(* CODESYS project cyber-gprs.lib.source.20190613.project

Project tree, tasks and I/O mapping:
  MIC7001 : Changsha Xiangji-ARM Cortex A9(xilinx zynq7000)-linux, Changsha Xiangji Hiden Technology Co.Ltd, version 3.5.10.40
    application Application
      libraries: CAA Types Extern, 3.5.10.0 (CAA Technical Workgroup); VisuDialogs, * (System); CAA Real Time Clock Extern, 3.5.10.0 (CAA Technical Workgroup); CAA Callback Extern, 3.5.11.0 (CAA Technical Workgroup); CAA Can Low Level Extern, 3.5.11.0 (CAA Technical Workgroup); CAA Can Low Level Imp Extern, 3.5.11.0 (CAA Technical Workgroup); SysMem, 3.5.12.0 (System); CAA Net Base Services, 3.5.12.0 (CAA Technical Workgroup); CAA SerialCom, 3.5.12.0 (CAA Technical Workgroup); CAA File, 3.5.12.0 (CAA Technical Workgroup); CAA DTUtil Extern, 3.5.12.0 (CAA Technical Workgroup); SysFile, 3.5.9.0 (System); SysTypes2 Interfaces, * (System); Standard, * (System); cyber gpio, 3.5.10.40 (cyber); Util, * (System)
      task Task_gprs (cyclic, interval 20 ms, priority 10) calls prg_heartbeat
      global variables GVL
      GPRS/
        function block File_Read [ST]
        function Iccid_Get [ST]
        program prg_heartbeat [ST]
        function block fb_get_iccid [ST]
        function block fb_m26 [ST]
        function block fb_get_lac [ST]
        function fn_cyber_layer1 [ST]
        function fn_cyber_layer2 [ST]
        function fn_cyber_heartBeat [ST]
        function fn_sn_str_to_byte [ST]
      gprs_lib/
        function block Com_Read [ST]
        function block reset_gprs [ST]
        function block Udp_Config [ST]
        function block Udp_Init [ST]
        function block UDP_Read [ST]
        function block Udp_Write [ST]
    IoDrvMIC7001 : IoDrvMIC7001, Cyber-MI, version 18.11.1
        unmapped channels: Ai00@C16, Ai01@C28, Ai02@C17, Ai03@C29, Ai04@C30, Ai05@C19, Ai06@C31, Ai07@C20, Ai08@C18, Ai09@D18, Ai10@D20, Ai11@D31, Ai12@D19, Ai13@D30, Ai14@D29, Ai15@D17, Ai16@D28, Ai17@D16, Ai18-Do00@C25, Ai19-Do01@C24, Ai20-Do02@C13, Ai21-Do03@C01, Ai22-Do04@C03, Ai23-Do05@C04, Ai24-Do06@C05, Ai25-Do07@C06, Ai26-Do08@C08, Ai27-Do09@C09, Ai28-Do10@C10, Ai29-Do11@C11, Ai30-Do12@D34, Ai31-Do13@D35, Ai32-Do14@D23, Ai33-Do15@D12, Ai34-Do16@D10, Ai35-Do17@D09, Ai36-Do18@D08, Ai37-Do19@D07, Ai38-Do20@D05, Ai39-Do21@D04,
          Ai40-Do22@D03, Ai41-Do23@D02, Ai42-Do24@C23, Ai43-Do25@C35, Ai44-Do26@D24, Ai45-Do27@D13, Ai46-Ao00@C22, Ai47-Ao01@D14, Ai48_Pi02, Ai49_Out5V, Ai50_VCC, Ai51_VCC_L, Ai52_VCC_R, Ai53_Pwm-i0, Ai54_Pwm-i1, Ai55_Pwm-i2, Ai56_Pwm-i3, Ai57_CPU-T, Ai58_G-x, Ai59_G-y, Ai60_G-z, Ai61-reserved, Ai62-IO-cntr, Ai63-CDS-cntr, Di00-Ai00@C16, Di01-Ai01@C28, Di02-Ai02@C17, Di03-Ai03@C29, Di04-Ai04@C30, Di05-Ai05@C19, Di06-Ai06@C31, Di07-Ai07@C20, Di08-Ai08@C18, Di09-Ai09@D18, Di10-Ai10@D20, Di11-Ai11@D31, Di12-Ai12@D19, Di13-Ai13@D30, Di14-Ai14@D29, Di15-Ai15@D17,
          Di16-Ai16@D28, Di17-Ai17@D16, Di18-Ai18@C25, Di19-Ai19@C24, Di20-Ai20@C13, Di21-Ai21@C01, Di22-Ai22@C03, Di23-Ai23@C04, Di24-Ai24@C05, Di25-Ai25@C06, Di26-Ai26@C08, Di27-Ai27@C09, Di28-Ai28@C10, Di29-Ai29@C11, Di30-Ai30@D34, Di31-Ai31@D35, Di32-Ai32@D23, Di33-Ai33@D12, Di34-Ai34@D10, Di35-Ai35@D09, Di36-Ai36@D08, Di37-Ai37@D07, Di38-Ai38@D05, Di39-Ai39@D04, Di40-Ai40@D03, Di41-Ai41@D02, Di42-Ai42@C23, Di43-Ai43@C35, Di44-Ai44@D24, Di45-Ai45@D13, Di46-Ai46@C22, Di47-Ai47@D14, Di48-Pi00@C15, Di49-Pi01@C14, Di50-Pi02@D22, Di51-Pi03@D21, Di52-reserved, Di53-reserved, Di54-reserved, Di55-reserved,
          Di56-reserved, Di57-reserved, Di58-reserved, Di59-reserved, Di60-reserved, Di61-reserved, Di62-reserved, Di63-reserved, Pi00-Di48@C15, Pi01-Di49@C14, Pi02-Di50@D22, Pi03-Di51@D21, Do00-Ai18@C25, Do01-Ai19@C24, Do02-Ai20@C13, Do03-Ai21@C01, Do04-Ai22@C03, Do05-Ai23@C04, Do06-Ai24@C05, Do07-Ai25@C06, Do08-Ai26@C08, Do09-Ai27@C09, Do10-Ai28@C10, Do11-Ai29@C11, Do12-Ai30@D34, Do13-Ai31@D35, Do14-Ai32@D23, Do15-Ai33@D12, Do16-Ai34@D10, Do17-Ai35@D09, Do18-Ai36@D08, Do19-Ai37@D07, Do20-Ai38@D05, Do21-Ai39@D04, Do22-Ai40@D03, Do23-Ai41@D02, Do24-Ai42@C23, Do25-Ai43@C35, Do26-Ai44@D24, Do27-Ai45@D13,
          Do28-Pwmi00@C33, Do29-Pwmi01@C34, Do30-Pwmi02@D25, Do31-Pwmi03@D26, PWM00@C25, PWM01@C24, PWM02@C13, PWM03@C01, PWM04@C03, PWM05@C04, PWM06@C05, PWM07@C06, PWM08@C08, PWM09@C09, PWM10@C10, PWM11@C11, PWM12@D34, PWM13@D35, PWM14@D23, PWM15@D12, PWM16@D10, PWM17@D09, PWM18@D08, PWM19@D07, PWM20@D05, PWM21@D04, PWM22@D03, PWM23@D02, PWM24@C23, PWM25@C35, PWM26@D24, PWM27@D13, PWM28-Pwmi00@C33, PWM29-Pwmi01@C34, PWM30-Pwmi02@D25, PWM31-Pwmi03@D26, PWM_I_0@C33, PWM_I_1@C34, PWM_I_2@D25, PWM_I_3@D26,
          Ao00-Ai46@C22, Ao01-Ai47@D14, LED_run, LED_err, LED_usr, ctrl_ai_raw, ctrl_adjust, ctrl_adj0, ctrl_adj1, ctrl_adj2, ctrl_adj3, ctrl_adj4
    SoftMotion General Axis Pool
  5ce3da45-db07-42e7-a21c-a00fff4ed8f6|C:\Users\Administrator\Desktop\robotview1.bmp
  5ce3da45-db07-42e7-a21c-a00fff4ed8f6|C:\Users\Administrator\Desktop\robotview2.bmp
  text list GlobalTextList
  5ce3da45-db07-42e7-a21c-a00fff4ed8f6|C:\Users\Administrator\Desktop\1129.bmp
  5ce3da45-db07-42e7-a21c-a00fff4ed8f6|C:\Users\Administrator\Desktop\robotview0.bmp
*)

// MIC7001/Application/GVL
VAR_GLOBAL
	
END_VAR

// MIC7001/Application/GPRS/prg_heartbeat
PROGRAM prg_heartbeat
VAR_OUTPUT
	lock_state :INT := 0;
	unlock_state :INT := 0;
	lock_unlock_level :INT := 0;
	delay_time :INT := 0;
END_VAR

VAR
	is_inited :BOOL := FALSE;
	g_m26:fb_m26;
	udp_handle :CAA.HANDLE; 
	udp_write_fb:Udp_Write;
	udp_read_fb:Udp_Read;
	file_read_fb:File_Read;
	com_read_fb :Com_Read;


	size :CAA.SIZE;	
	Writebuffer: 			ARRAY[1..200] OF BYTE;
	Readbuffer: 			ARRAY[0..1499] OF BYTE;
	ReadbufferStr: STRING;
	atcState :INT := 0;
	
	writeUdpState :INT := 0;
	readUdpState :INT := 0;
	
	i :INT;
	count :INT := 0;
	
	rtc_fb: RTC;
	dtu_set_dt_fb: dtu.SetDateAndTime;
	
	sn_file_name :STRING := '/userapp/sn.txt';
	time_file_name :STRING := '/userapp/r_mins.txt';
	is_read :BOOL := FALSE;
	read_count :INT := 0;
	readFileState :INT := 0;
	ton_fb :TON;
	iccid_read_buffer :STRING;
	position :INT := -1;
	new_date:DT;
	get_iccid:fb_get_iccid;
	get_lac:fb_get_lac;
	iStat :UINT := 0;
	lac : STRING(4) := '0000';
	ci : STRING(4) := '0000';
	lenHearBeat:UINT;
	dataHearBeat:ARRAY[0..255] OF BYTE;
	ton_hb:ton; //heartbeat timer 
	bReturn:BOOL;
	lenLayer2:UINT;
	dataLayer2:ARRAY[0..255] OF BYTE;
	lenLayer1:UINT;
	lenRecvLayer1:UINT := 1500;
	dataLayer1:ARRAY[0..255] OF BYTE;
	bSN :ARRAY[0..6] OF BYTE;
	sub_str:STRING(8);
	num :UINT;
	lenHeartBeat: UINT;
	sn: STRING;
	work_time: UDINT;
	dataIndex :UINT := 0;
	cntr_lac:UINT := 0;
	cntr_iccid:UINT := 0;
	
	recv_size :CAA.SIZE;
END_VAR

CASE iStat OF
0:
	g_m26(enable := TRUE, ipaddr := '47.107.240.29', port := 20861);  //共用的基础模块，只要有一个地方调用即可	
	IF g_m26.xDone THEN
		iStat := 1;
	END_IF


1:  // read iccid
	get_iccid(xExecute := FALSE);
	iStat := 2;
	cntr_iccid := 0;
	
2:
	get_iccid(xExecute := TRUE, m26_handle := g_m26.handle_m26);
	IF get_iccid.xDone THEN
		iccid_read_buffer := get_iccid.iccid;
		iStat := 10;
	END_IF
	cntr_iccid := cntr_iccid + 1;
	IF cntr_iccid > 600 THEN   // 1 min
		iStat := 1;
	END_IF
	
10: //read sn
	file_read_fb(file_name := sn_file_name);
	IF file_read_fb.isRead THEN
		sn := file_read_fb.sReadLine;
		iStat := 15;
	END_IF
	
15:
	get_lac(xExecute := FALSE);	
	iStat := 20;
	cntr_lac := 0;
	
20:
	get_lac(xExecute := TRUE, m26_handle := g_m26.handle_m26);
	IF get_lac.xDone THEN
		lac := get_lac.lac;
		ci := get_lac.ci;
		iStat := 30;
	END_IF
	cntr_lac := cntr_lac + 1;
	IF cntr_lac > 200 THEN
		iStat := 0;
	END_IF
	
30:
	file_read_fb(file_name := time_file_name);
	IF file_read_fb.isRead THEN
		work_time := STRING_TO_UDINT(file_read_fb.sReadLine);
		iStat := 100;
	END_IF
	
100:
	ton_fb(IN := TRUE, PT := T#60S);
	IF (ton_fb.Q) THEN
		ton_fb(IN := FALSE, PT := T#60S);
		iStat := 200;
	END_IF
	
200:
	bReturn := fn_cyber_heartBeat(	  //填充第三层：心跳帧
						lac_str := lac, 
						cid_str := ci, 
						ccid_str := iccid_read_buffer, 
						mins := work_time, 
						clientCode := 1, 
						machineCode := 1, 
						pLenOut := ADR(lenHearBeat), 
						pDataOut := ADR(dataHearBeat));
	IF NOT bReturn THEN
		RETURN;
	ELSE
		iStat := 300;
	END_IF;

300:
	dataIndex := dataIndex + 1;
	bReturn := fn_cyber_layer2( //填充第二层，数据层
						dataType := 1,
						paraId := 0,
						dataIndex := dataIndex,
						ver := 1,
						res1 := 0,
						LenIn := lenHearBeat,
						pDataIn := ADR(dataHearBeat),
						pLenOut := ADR(lenLayer2),
						pDataOut := ADR(dataLayer2));
						
	IF NOT bReturn THEN
		RETURN;
	ELSE
		iStat := 400;
	END_IF;
	
400:
	bSN := fn_sn_str_to_byte(sn);
	bReturn := fn_cyber_layer1(    //填充第一层，设备层
						sn := ADR(bSN),
						ver := 1,
						lenIn := lenLayer2,
						pDataIn := ADR(dataLayer2),
						pLenOut := ADR(lenLayer1),
						pDataOut := ADR(dataLayer1));
	IF NOT bReturn THEN
		RETURN;
	ELSE
		udp_write_fb(xExecute := FALSE);
		iStat := 500;
	END_IF;
		
	
500:
	udp_write_fb(xExecute := TRUE, com := g_m26.handle_m26, buffer := ADR(dataLayer1), size := lenLayer1);
	IF udp_write_fb.xDone THEN
		udp_write_fb(xExecute := FALSE);
		udp_read_fb(xExecute := FALSE);
		iStat := 600; 
	END_IF
	
	IF udp_write_fb.xError THEN  
		udp_write_fb(xExecute := FALSE);
		iStat := 15; 
	END_IF
	
	
600:
	udp_read_fb(xExecute := TRUE, com := g_m26.handle_m26, buffer := ADR(Readbuffer), rsize := sizeof(Readbuffer));
	IF udp_read_fb.xDone THEN  //接收到数据
	 	recv_size := udp_read_fb.size;
		udp_read_fb(xExecute := FALSE);
		iStat := 15; //read mins and lca again
		IF recv_size = 26 THEN
			lock_state := BYTE_TO_INT(Readbuffer[20]);
			unlock_state := BYTE_TO_INT(Readbuffer[21]);
			lock_unlock_level := BYTE_TO_INT(Readbuffer[22]);
			delay_time := BYTE_TO_INT(Readbuffer[23]);
		END_IF
	END_IF
	
	IF udp_read_fb.xError THEN  //接收到数据
		udp_read_fb(xExecute := FALSE);
		recv_size := 0;
		iStat := 15; //read mins and lca again
	END_IF

END_CASE

RETURN;

END_PROGRAM

// MIC7001/Application/GPRS/fn_cyber_heartBeat
FUNCTION fn_cyber_heartBeat : bool
VAR_INPUT
	lac_str:STRING(4);
	cid_str:STRING(4);
	ccid_str:STRING(21);
	mins:UDINT;
	clientCode:UINT;
	machineCode:UINT;
	pLenOut:POINTER TO UINT;
	pDataOut:POINTER TO BYTE;
END_VAR
VAR
	index: UINT;
	data_uint: UINT;
	data_byte_array:ARRAY[0..9] OF BYTE;
	i: INT;
END_VAR

fn_cyber_heartBeat := FALSE;

index := 0;
data_uint := STRING_TO_UINT(concat('16#',lac_str));
pDataOut[index] := ANY_TO_BYTE(data_uint/256);
index := index + 1;

pDataOut[index] := ANY_TO_BYTE(data_uint MOD 256);
index := index + 1;

data_uint := STRING_TO_UINT(concat('16#',cid_str));
pDataOut[index] := ANY_TO_BYTE(data_uint/256);
index := index + 1;

pDataOut[index] := ANY_TO_BYTE(data_uint MOD 256);
index := index + 1;

data_byte_array := Iccid_Get(ccid_str);
FOR i := 0 TO 9 DO
	pDataOut[index] := data_byte_array[i];
	index := index + 1;
END_FOR

pDataOut[index] := ANY_TO_BYTE(mins/256/256/256);
index := index + 1;

pDataOut[index] := ANY_TO_BYTE(mins/256/256);
index := index + 1;

pDataOut[index] := ANY_TO_BYTE(mins/256);
index := index + 1;

pDataOut[index] := ANY_TO_BYTE(mins);
index := index + 1;

pDataOut[index] := ANY_TO_BYTE(clientCode/256);
index := index + 1;

pDataOut[index] := ANY_TO_BYTE(clientCode);
index := index + 1;

pDataOut[index] := ANY_TO_BYTE(machineCode/256);
index := index + 1;

pDataOut[index] := ANY_TO_BYTE(machineCode);
index := index + 1;

pLenOut^ := index;

fn_cyber_heartBeat := TRUE;

END_FUNCTION

// MIC7001/Application/GPRS/Iccid_Get
FUNCTION Iccid_Get : ARRAY[0..9] OF BYTE
VAR_INPUT
	iccd :STRING;
END_VAR
VAR
	iccid_code :ARRAY[0..9] OF BYTE;
	
	byteHigh :BYTE := 0;
	byteLow :BYTE := 0;
	dstLen :INT := 0;
	
	srcIndex :INT := 0;
	bytesIndex :INT := 0;
	sub_str:STRING(32);
END_VAR

dstLen := len(iccd) / 2;

sub_str := iccd;
FOR bytesIndex := 0 TO dstLen - 1 DO
	iccid_code[bytesIndex] := BYTE_TO_BCD(STRING_TO_BYTE(left(sub_str,2)));	
	sub_str := delete(sub_str,2,1);
END_FOR

Iccid_Get := iccid_code;

END_FUNCTION

// MIC7001/Application/GPRS/fn_cyber_layer2
FUNCTION fn_cyber_layer2 : bool
VAR_INPUT
	dataType : BYTE := 0;
	paraId :BYTE := 0;
	dataIndex : UINT := 0;
	ver :BYTE := 1;
	res1 :BYTE := 0;
	LenIn :UINT := 0;
	pDataIn :POINTER TO BYTE;
	pLenOut :POINTER TO UINT;
	pDataOut :POINTER TO BYTE;
END_VAR
VAR
	i:UINT:= 0;
	index:UINT := 0;
END_VAR

fn_cyber_layer2 := FALSE;

index := 0;
pDataOut[index] := dataType;
index := index + 1;

pDataOut[index] := paraId;
index := index + 1;

pDataOut[index] := ANY_TO_BYTE(dataIndex/256);
index := index + 1;

pDataOut[index] := ANY_TO_BYTE(dataIndex MOD 256);
index := index + 1;

pDataOut[index] := ver;
index := index + 1;

pDataOut[index] := res1;
index := index + 1;

pDataOut[index] := ANY_TO_BYTE(LenIn/256);
index := index + 1;

pDataOut[index] := ANY_TO_BYTE(LenIn MOD 256);
index := index + 1;

FOR i := 0 TO LenIn-1 DO
	pDataOut[index] := pDataIn[i];
	index := index + 1;
END_FOR

pLenOut^ := index;

fn_cyber_layer2 := TRUE;
RETURN;

END_FUNCTION

// MIC7001/Application/GPRS/fn_sn_str_to_byte
FUNCTION fn_sn_str_to_byte : ARRAY[0..6] OF BYTE
VAR_INPUT
	sn:STRING(16);
END_VAR
VAR
	i: INT;
	bSN: ARRAY[0..6] OF BYTE;
	sub_str: STRING(255);
	num: UINT;
	bcd: UINT;
END_VAR

// 1.2 12
sub_str := mid(sn, 2, 4);
bcd := STRING_TO_UINT(sub_str);
bcd := (bcd / 10) *16 + (bcd MOD 10);
bSN[0] := UINT_TO_BYTE(bcd);

// 1.3 34
sub_str := mid(sn, 2, 6);
bcd := STRING_TO_UINT(sub_str);
bcd := (bcd / 10) *16 + (bcd MOD 10);
bSN[1] := UINT_TO_BYTE(bcd);

// 1.4 56
sub_str := mid(sn, 2, 8);
bcd := STRING_TO_UINT(sub_str);
bcd := (bcd / 10) *16 + (bcd MOD 10);
bSN[2] := UINT_TO_BYTE(bcd);

// 1.5 78
sub_str := mid(sn, 2, 10);
bcd := STRING_TO_UINT(sub_str);
bcd := (bcd / 10) *16 + (bcd MOD 10);
bSN[3] := UINT_TO_BYTE(bcd);

// 1.6 1234
sub_str := mid(sn, 2, 12);
bcd := STRING_TO_UINT(sub_str);
bcd := (bcd / 10) *16 + (bcd MOD 10);
bSN[4] := UINT_TO_BYTE(bcd);

sub_str := mid(sn, 2, 14);
bcd := STRING_TO_UINT(sub_str);
bcd := (bcd / 10) *16 + (bcd MOD 10);
bSN[5] := UINT_TO_BYTE(bcd);

fn_sn_str_to_byte := bSN;

END_FUNCTION

// MIC7001/Application/GPRS/fn_cyber_layer1
FUNCTION fn_cyber_layer1 : bool
VAR_INPUT
	sn:POINTER TO BYTE;
	ver:BYTE := 0;
	lenIn:UINT := 0;
	pDataIn:POINTER TO BYTE;
	pLenOut:POINTER TO UINT ;
	pDataOut: POINTER TO BYTE;
END_VAR
VAR
	i:UINT;
	index:UINT;
	checksum:UINT;
	res1 :BYTE := 0;
	res2 :BYTE := 0;
	res3 :BYTE := 0;
END_VAR

fn_cyber_layer1 := FALSE;

index := 0;
checksum := 0;
FOR i := 0 TO 5 DO
	pDataOut[index] := sn[i];
	index := index+1;
	checksum := checksum + sn[i];
END_FOR

pDataOut[index] := ver;
index := index+1;
checksum := checksum + ver;

pDataOut[index] := res1;
index := index+1;
checksum := checksum + res1;

pDataOut[index] := res2;
index := index+1;
checksum := checksum + res2;

pDataOut[index] := res3;
index := index+1;
checksum := checksum + res3;

pDataOut[index] := ANY_TO_BYTE(lenIn/256);
index := index+1;
checksum := checksum + ANY_TO_BYTE(lenIn/256);

pDataOut[index] := ANY_TO_BYTE(lenIn MOD 256);
index := index+1;
checksum := checksum + ANY_TO_BYTE(lenIn MOD 256);

FOR i := 0 TO lenIn-1 DO
	pDataOut[index] := pDataIn[i];
	index := index+1;	
	checksum := checksum + pDataIn[i];
END_FOR

pDataOut[index] := ANY_TO_BYTE(checksum/256);
index := index+1;

pDataOut[index] := ANY_TO_BYTE(checksum MOD 256);
index := index+1;

pLenOut^ := index;

fn_cyber_layer1 := TRUE;

END_FUNCTION

// MIC7001/Application/GPRS/fb_m26
FUNCTION_BLOCK fb_m26
VAR_INPUT
	enable :BOOL := FALSE;
	ipaddr :STRING(32);
	port :UINT;
END_VAR
VAR_OUTPUT
	xBusy :BOOL := FALSE;
	xError :BOOL := FALSE;
	xDone :BOOL := FALSE;
	handle_m26 :CAA.HANDLE; 
END_VAR
VAR
	udp_init:Udp_Init;
	iStat :UINT := 0;
END_VAR

IF NOT enable THEN
	xBusy := FALSE;
	xError := FALSE;
	handle_m26 := 0;
	RETURN;
END_IF

CASE iStat OF
0:
	udp_init(xExecute := FALSE, ip_addr := ipaddr, port := port);
	udp_init.xExecute := TRUE;
	iStat := 10;
	
10:
	IF udp_init.xDone THEN
		xBusy := TRUE;
		handle_m26 := udp_init.udp_handle;
		iStat := 100;
	ELSIF udp_init.xError THEN
		iStat := 200;
	END_IF	

100:
	xDone:= TRUE;
	
200:
	xError := TRUE;

END_CASE


udp_init(ip_addr := ipaddr, port := port);

END_FUNCTION_BLOCK

// MIC7001/Application/gprs_lib/Udp_Init
FUNCTION_BLOCK Udp_Init
VAR_INPUT
	xExecute:BOOL := FALSE;
	ip_addr:STRING;
	port:UINT;
END_VAR
VAR_OUTPUT
	xDone :BOOL := FALSE;
	xError :BOOL := FALSE;
	xBusy :BOOL := FALSE;
	
	udp_handle :CAA.HANDLE; 
END_VAR
VAR
	udp_config_fb :Udp_Config;
	ComWrite: COM.Write;
	ComRead: COM.Read;	
	com_handle: CAA.HANDLE;
	init_start :DWORD := 0;
	iStat: INT := 0;
END_VAR

init_start := %ID48;
IF (init_start > 0) THEN
	RETURN;
END_IF

IF NOT xExecute THEN
	xDone := FALSE;
	xError := FALSE;
	xBusy := FALSE;
	iStat := 0;
	RETURN;
END_IF

CASE iStat OF
0:
	udp_config_fb(xExecute := FALSE,ip_addr := ip_addr, port := port, com_hand := com_handle); 
	iStat := 10;
	xBusy := TRUE;
10:
	udp_config_fb.xExecute := TRUE;
	IF udp_config_fb.xDone  THEN
		iStat := 100;
		xDone := TRUE;
		xBusy := FALSE;
		udp_handle := com_handle;
		ComWrite(xExecute := FALSE, hCom:= com_handle);
		ComRead(xExecute := FALSE, hCom:= com_handle);		
	ELSIF udp_config_fb.xError THEN
		xError := TRUE;
		iStat := 200;
	END_IF	
100: //succ

200: //error

END_CASE

udp_config_fb(ip_addr := ip_addr, port := port, com_hand := com_handle);

END_FUNCTION_BLOCK

// MIC7001/Application/gprs_lib/Udp_Config
FUNCTION_BLOCK Udp_Config
VAR_INPUT
	xExecute : BOOL := FALSE;
	ip_addr:STRING;
	port:UINT;
END_VAR
VAR_IN_OUT
	com_hand: CAA.HANDLE;
END_VAR
VAR_OUTPUT
	xDone : BOOL := FALSE;
	xError :BOOL := FALSE;
	xBusy : BOOL := FALSE;
END_VAR
VAR
	ton_fb :TON;
	Com1Params: 			ARRAY [1..7] OF COM.PARAMETER;	(* Settings to communicate with 
the COM Port *)
	ComOpen: 				COM.Open;
	ComClose: 				COM.Close;
	ComWrite: 				COM.Write;
	ComRead: 				COM.Read;	
	Rcv_Cnt: 				CAA.SIZE;
	xCom1CloseError: 		BOOL;
	xCom1WriteError: 		BOOL;
	xCom1ReadError: 		BOOL;
	uiComState: INT := 0;
	ComID:USINT:=6;

	position :INT := 0;
	at_cmd :STRING := 'AT$r';
	at_buffer :STRING;
	ate0_cmd :STRING := 'ATE0$r';
	ate0_buffer :STRING;
	cpin_cmd :STRING := 'AT+CPIN?$r';
	cpin_buffer :STRING;
	csq_cmd :STRING := 'AT+CSQ$r';
	csq_buffer :STRING;
	creg_cmd :STRING := 'AT+CREG?$r';
	creg_buffer :STRING;
	cgreg_cmd :STRING := 'AT+CGREG?$r';
	cgreg_buffer :STRING;
	qindi_cmd :STRING := 'AT+QINDI=1$r';
	qindi_buffer :STRING;     
	qimode_cmd :STRING := 'AT+QIMODE=0$r';
	qimode_buffer :STRING;     
	qifgcnt_cmd :STRING := 'AT+QIFGCNT=0$r';
	qifgcnt_buffer :STRING;
	qimux_cmd :STRING := 'AT+QIMUX=0$r';
	qimux_buffer :STRING;
	qicsgp_cmd :STRING := 'AT+QICSGP=1,$"CMNET$"$r';
	qicsgp_buffer :STRING;
	qideact_cmd :STRING := 'AT+QIDEACT$r';
	qideact_buffer :STRING;
	qiregapp_cmd :STRING := 'AT+QIREGAPP$r';
	qiregapp_buffer :STRING;
	qiact_cmd :STRING := 'AT+QIACT$r';
	qiact_buffer :STRING;
	qilocip_cmd :STRING := 'AT+QILOCIP$r';
	qilocip_buffer :STRING;
	qiopen_cmd :STRING := 'AT+QIOPEN=$"UDP$",$"';
	qiopen_buffer :STRING;
	
	qntp_cmd: STRING := 'AT+QNTP=$"s1a.time.edu.cn$"$r';
	qntp_buffer: STRING;
	qnitz_cmd: STRING := 'AT+QNITZ=1$r';	//启用同步网络时间
	qnitz_buffer :STRING;
	ctzu_cmd: STRING := 'AT+CTZU=1$r';
	ctzu_buffer: STRING;
	qlts_cmd: STRING := 'AT+QLTS$r';
	qlts_buffer: STRING;
	cclk_cmd: STRING := 'AT+CCLK?$r';
	cclk_buffer: STRING;
	
	NewDT : DT;
	NewDTS : STRING;
	NewDTSZH : STRING;
	dtu_set_dt_fb: dtu.SetDateAndTime;
	dtu_set_zone_fb: dtu.SetTimeZoneInformation;
	zone: RTCLK.TIME_ZONE_INFO;
	year: int;
	
	//dtu_get_zone_fb: dtu.GetTimeZoneInformation;
	//zone1: RTCLK.TIME_ZONE_INFO;

	loop_in_count :INT := 0;
	loop_out_count :INT := 0;
	loop_count :INT := 0;
	connect_cnt :INT := 0;
	reset_gprs_fb :reset_gprs;
END_VAR

IF NOT xExecute THEN
	xDone := FALSE;
	xError := FALSE;
	xBusy := FALSE;
	uiComState := 0;
	RETURN;
END_IF

CASE uiComState OF
	0:
	Com1Params[1].udiParameterId := COM.CAA_Parameter_Constants.udiPort;
	Com1Params[1].udiValue := ComID; 
	Com1Params[2].udiParameterId := COM.CAA_Parameter_Constants.udiBaudrate;
	Com1Params[2].udiValue := 115200;
	Com1Params[3].udiParameterId := COM.CAA_Parameter_Constants.udiParity;
	Com1Params[3].udiValue := INT_TO_UINT(COM.PARITY.NONE);
	Com1Params[4].udiParameterId := COM.CAA_Parameter_Constants.udiStopBits;
	Com1Params[4].udiValue := INT_TO_UINT(COM.STOPBIT.ONESTOPBIT);
	Com1Params[5].udiParameterId := COM.CAA_Parameter_Constants.udiTimeout;
	Com1Params[5].udiValue := 0;
	Com1Params[6].udiParameterId := COM.CAA_Parameter_Constants.udiByteSize;
	Com1Params[6].udiValue := 8;
	Com1Params[7].udiParameterId := COM.CAA_Parameter_Constants.udiBinary;
	Com1Params[7].udiValue := 0;					
	ComOpen(xExecute := TRUE, usiListLength:=UINT_TO_USINT(SIZEOF(Com1Params)/SIZEOF(COM.PARAMETER)),pParameterList:= ADR(Com1Params),hCom=> com_hand);			
	IF ComOpen.xError THEN
		uiComState := 32767;
	ELSIF ComOpen.xDone THEN
		uiComState := 1;
		com_hand := ComOpen.hCom;
		ComWrite(xExecute := FALSE,hCom:= com_hand);	
		ComRead(xExecute := FALSE,hCom:= com_hand);
	END_IF
	
	1:  // write "AT\r"
	ComWrite(xExecute := TRUE,hCom:= com_hand,pBuffer:= ADR(at_cmd),szSize:=len(at_cmd));		
	IF ComWrite.xError THEN
		uiComState := 32767;
	END_IF
	IF ComWrite.xDone THEN
		ComWrite(xExecute := FALSE, hCom:= com_hand);
		uiComState := 2;
	END_IF
	
	2:
	ton_fb(IN := TRUE, PT := TIME#300MS);
	IF (ton_fb.Q) THEN
		ton_fb(IN := FALSE, PT := TIME#300MS);
		uiComState := 3;
	END_IF
	
	3:
	ComRead(xExecute := TRUE,hCom:= com_hand, pBuffer:= ADR(at_buffer), szBuffer:= SIZEOF(at_buffer));			
	IF ComRead.xError THEN
		uiComState := 32767;
	END_IF
	IF ComRead.xDone THEN
		uiComState := 1;
		position := find(at_buffer, 'OK');
		IF position > 0 THEN
			uiComState := 4;
			loop_in_count := 0;
			loop_out_count := 0;
		END_IF
		ComRead(xExecute := FALSE, hCom:= com_hand);
	
		IF loop_out_count > 10 THEN
			uiComState := 32767;
			RETURN;
		END_IF
		
		// 通过gpio复位gprs模块
		loop_in_count := loop_in_count + 1;
		IF loop_in_count > 50 THEN
			loop_in_count := 0;
			loop_out_count := loop_out_count + 1;
			reset_gprs_fb(xExecute := FALSE);
			uiComState := 250;
			RETURN;
		END_IF
	END_IF
		
	4: // write "ATE0\r"
	ComWrite(xExecute := TRUE,hCom:= com_hand,pBuffer:= ADR(ate0_cmd),szSize:=len(ate0_cmd));		
	IF ComWrite.xError THEN
		uiComState := 32767;
	END_IF
	IF ComWrite.xDone THEN
		ComWrite(xExecute := FALSE, hCom:= com_hand);
		uiComState := 5;
	END_IF
	
	5:
	ton_fb(IN := TRUE, PT := TIME#300MS);
	IF (ton_fb.Q) THEN
		ton_fb(IN := FALSE, PT := TIME#300MS);
		uiComState := 6;
	END_IF
	
	6:
	ComRead(xExecute := TRUE,hCom:= com_hand, pBuffer:= ADR(ate0_buffer), szBuffer:= SIZEOF(ate0_buffer));			
	IF ComRead.xError THEN
		uiComState := 32767;
	END_IF
	IF ComRead.xDone THEN
		uiComState := 4;
		ComRead(xExecute := FALSE, hCom:= com_hand);
		position := find(ate0_buffer, 'OK');
		IF position > 0 THEN
			uiComState := 7;
		END_IF
	END_IF
	
	7: // write "AT+CPIN?\r"
	ComWrite(xExecute := TRUE,hCom:= com_hand,pBuffer:= ADR(cpin_cmd),szSize:=len(cpin_cmd));		
	IF ComWrite.xError THEN
		uiComState := 32767;
	END_IF
	IF ComWrite.xDone THEN
		ComWrite(xExecute := FALSE, hCom:= com_hand);
		uiComState := 8;
	END_IF
	
	8:
	ton_fb(IN := TRUE, PT := TIME#300MS);
	IF (ton_fb.Q) THEN
		ton_fb(IN := FALSE, PT := TIME#300MS);
		uiComState := 9;
	END_IF
	
	9:
	ComRead(xExecute := TRUE,hCom:= com_hand, pBuffer:= ADR(cpin_buffer), szBuffer:= SIZEOF(cpin_buffer));			
	IF ComRead.xError THEN
		uiComState := 32767;
	END_IF
	IF ComRead.xDone THEN
		uiComState := 7;
		ComRead(xExecute := FALSE, hCom:= com_hand);
		position := find(cpin_buffer, 'OK');
		IF position > 0 THEN
			uiComState := 10;
		END_IF
	END_IF
	
	10: // write "AT+CSQ\r"
	ComWrite(xExecute := TRUE,hCom:= com_hand,pBuffer:= ADR(csq_cmd),szSize:=len(csq_cmd));		
	IF ComWrite.xError THEN
		uiComState := 32767;
	END_IF
	IF ComWrite.xDone THEN
		ComWrite(xExecute := FALSE, hCom:= com_hand);
		uiComState := 11;
	END_IF
	
	11:
	ton_fb(IN := TRUE, PT := TIME#300MS);
	IF (ton_fb.Q) THEN
		ton_fb(IN := FALSE, PT := TIME#300MS);
		uiComState := 12;
	END_IF
	
	12:
	ComRead(xExecute := TRUE,hCom:= com_hand, pBuffer:= ADR(csq_buffer), szBuffer:= SIZEOF(csq_buffer));			
	IF ComRead.xError THEN
		uiComState := 32767;
	END_IF
	IF ComRead.xDone THEN
		uiComState := 10;
		ComRead(xExecute := FALSE, hCom:= com_hand);
		position := find(csq_buffer, 'OK');
		IF position > 0 THEN
			uiComState := 13;
		END_IF
	END_IF
	
	13: // write "AT+CREG?\r"
	ComWrite(xExecute := TRUE,hCom:= com_hand,pBuffer:= ADR(creg_cmd),szSize:=len(creg_cmd));		
	IF ComWrite.xError THEN
		uiComState := 32767;
	END_IF
	IF ComWrite.xDone THEN
		ComWrite(xExecute := FALSE, hCom:= com_hand);
		uiComState := 14;
	END_IF
	
	14:
	ton_fb(IN := TRUE, PT := TIME#300MS);
	IF (ton_fb.Q) THEN
		ton_fb(IN := FALSE, PT := TIME#300MS);
		uiComState := 15;
	END_IF
	
	15:
	ComRead(xExecute := TRUE,hCom:= com_hand, pBuffer:= ADR(creg_buffer), szBuffer:= SIZEOF(creg_buffer));			
	IF ComRead.xError THEN
		uiComState := 32767;
	END_IF
	IF ComRead.xDone THEN
		uiComState := 13;
		ComRead(xExecute := FALSE, hCom:= com_hand);
		position := find(creg_buffer, 'OK');
		IF position > 0 THEN
			uiComState := 16;
		END_IF
	END_IF
	
	16: // write "AT+CGREG?\r"
	ComWrite(xExecute := TRUE,hCom:= com_hand,pBuffer:= ADR(cgreg_cmd),szSize:=len(cgreg_cmd));		
	IF ComWrite.xError THEN
		uiComState := 32767;
	END_IF
	IF ComWrite.xDone THEN
		ComWrite(xExecute := FALSE, hCom:= com_hand);
		uiComState := 17;
	END_IF
	
	17:
	ton_fb(IN := TRUE, PT := TIME#300MS);
	IF (ton_fb.Q) THEN
		ton_fb(IN := FALSE, PT := TIME#300MS);
		uiComState := 18;
	END_IF
	
	18:
	ComRead(xExecute := TRUE,hCom:= com_hand, pBuffer:= ADR(cgreg_buffer), szBuffer:= SIZEOF(cgreg_buffer));			
	IF ComRead.xError THEN
		uiComState := 32767;
	END_IF
	IF ComRead.xDone THEN
		uiComState := 16;
		ComRead(xExecute := FALSE, hCom:= com_hand);
		position := find(cgreg_buffer, 'OK');
		IF position > 0 THEN
			uiComState := 19;
		END_IF
	END_IF
	
	19: // write "AT+QINDI=1\r"     
	ComWrite(xExecute := TRUE,hCom:= com_hand,pBuffer:= ADR(qindi_cmd),szSize:=len(qindi_cmd));		
	IF ComWrite.xError THEN
		uiComState := 32767;
	END_IF
	IF ComWrite.xDone THEN
		ComWrite(xExecute := FALSE, hCom:= com_hand);
		uiComState := 20;
	END_IF
	
	20:
	ton_fb(IN := TRUE, PT := TIME#300MS);
	IF (ton_fb.Q) THEN
		ton_fb(IN := FALSE, PT := TIME#300MS);
		uiComState := 21;
	END_IF
	
	21:
	ComRead(xExecute := TRUE,hCom:= com_hand, pBuffer:= ADR(qindi_buffer), szBuffer:= SIZEOF(qindi_buffer));			
	IF ComRead.xError THEN
		uiComState := 32767;
	END_IF
	IF ComRead.xDone THEN
		uiComState := 19;
		ComRead(xExecute := FALSE, hCom:= com_hand);
		position := find(qindi_buffer, 'OK');
		IF position > 0 THEN
			uiComState := 22;
			loop_in_count := 0;
			loop_out_count := 0;
		ELSE
			IF loop_out_count > 10 THEN
				uiComState := 32767;
				RETURN;
			END_IF
			
			// 通过gpio复位gprs模块
			loop_in_count := loop_in_count + 1;
			IF loop_in_count > 25 THEN
				loop_in_count := 0;
				loop_out_count := loop_out_count + 1;
				reset_gprs_fb(xExecute := FALSE);
				uiComState := 250;
				RETURN;
			END_IF
		END_IF
	END_IF
	
	22: // write "AT+QIMODE=0\r"     
	ComWrite(xExecute := TRUE,hCom:= com_hand,pBuffer:= ADR(qimode_cmd),szSize:=len(qimode_cmd));		
	IF ComWrite.xError THEN
		uiComState := 32767;
	END_IF
	IF ComWrite.xDone THEN
		ComWrite(xExecute := FALSE, hCom:= com_hand);
		uiComState := 23;
	END_IF
	
	23:
	ton_fb(IN := TRUE, PT := TIME#300MS);
	IF (ton_fb.Q) THEN
		ton_fb(IN := FALSE, PT := TIME#300MS);
		uiComState := 24;
	END_IF
	
	24:
	ComRead(xExecute := TRUE,hCom:= com_hand, pBuffer:= ADR(qimode_buffer), szBuffer:= SIZEOF(qimode_buffer));			
	IF ComRead.xError THEN
		uiComState := 32767;
	END_IF
	IF ComRead.xDone THEN
		uiComState := 22;
		ComRead(xExecute := FALSE, hCom:= com_hand);
		position := find(qimode_buffer, 'OK');
		IF position > 0 THEN
			uiComState := 25;
		ELSE
			IF loop_out_count > 10 THEN
				uiComState := 32767;
				RETURN;
			END_IF
			
			// 通过gpio复位gprs模块
			loop_in_count := loop_in_count + 1;
			IF loop_in_count > 25 THEN
				loop_in_count := 0;
				loop_out_count := loop_out_count + 1;
				reset_gprs_fb(xExecute := FALSE);
				uiComState := 250;
				RETURN;
			END_IF
		END_IF
		//uiComState := 25;
	END_IF
	
	25: // write "AT+QIFGCNT=0\r"     
	ComWrite(xExecute := TRUE,hCom:= com_hand,pBuffer:= ADR(qifgcnt_cmd),szSize:=len(qifgcnt_cmd));		
	IF ComWrite.xError THEN
		uiComState := 32767;
	END_IF
	IF ComWrite.xDone THEN
		ComWrite(xExecute := FALSE, hCom:= com_hand);
		uiComState := 26;
	END_IF
	
	26:
	ton_fb(IN := TRUE, PT := TIME#300MS);
	IF (ton_fb.Q) THEN
		ton_fb(IN := FALSE, PT := TIME#300MS);
		uiComState := 27;
	END_IF
	
	27:
	ComRead(xExecute := TRUE,hCom:= com_hand, pBuffer:= ADR(qifgcnt_buffer), szBuffer:= SIZEOF(qifgcnt_buffer));			
	IF ComRead.xError THEN
		uiComState := 32767;
	END_IF
	IF ComRead.xDone THEN
		uiComState := 25;
		ComRead(xExecute := FALSE, hCom:= com_hand);
		position := find(qifgcnt_buffer, 'OK');
		IF position > 0 THEN
			uiComState := 28;
			loop_count := 0;
		END_IF
	END_IF
	
	28: // write "AT+QIMUX=0\r"     
	ComWrite(xExecute := TRUE,hCom:= com_hand,pBuffer:= ADR(qimux_cmd),szSize:=len(qimux_cmd));		
	IF ComWrite.xError THEN
		uiComState := 32767;
	END_IF
	IF ComWrite.xDone THEN
		ComWrite(xExecute := FALSE, hCom:= com_hand);
		uiComState := 29;
	END_IF
	
	29:
	ton_fb(IN := TRUE, PT := TIME#300MS);
	IF (ton_fb.Q) THEN
		ton_fb(IN := FALSE, PT := TIME#300MS);
		uiComState := 30;
	END_IF
	
	30:
	ComRead(xExecute := TRUE,hCom:= com_hand, pBuffer:= ADR(qimux_buffer), szBuffer:= SIZEOF(qimux_buffer));			
	IF ComRead.xError THEN
		uiComState := 32767;
	END_IF
	IF ComRead.xDone THEN
		uiComState := 28;
		ComRead(xExecute := FALSE, hCom:= com_hand);
		position := find(qimux_buffer, 'OK');
		IF position > 0 THEN
			uiComState := 31;
		END_IF
		//uiComState := 31;
		
		loop_count := loop_count + 1;
		IF loop_count > 100 THEN
			loop_count := 0;
			reset_gprs_fb(xExecute := FALSE);
			uiComState := 250;
			RETURN;
		END_IF
	END_IF
	
	31: // write "AT+QICSGP=1,\"CMNET\"\r"     
	ComWrite(xExecute := TRUE,hCom:= com_hand,pBuffer:= ADR(qicsgp_cmd),szSize:=len(qicsgp_cmd));		
	IF ComWrite.xError THEN
		uiComState := 32767;
	END_IF
	IF ComWrite.xDone THEN
		ComWrite(xExecute := FALSE, hCom:= com_hand);
		uiComState := 32;
	END_IF
	
	32:
	ton_fb(IN := TRUE, PT := TIME#300MS);
	IF (ton_fb.Q) THEN
		ton_fb(IN := FALSE, PT := TIME#300MS);
		uiComState := 33;
	END_IF
	
	33:
	ComRead(xExecute := TRUE,hCom:= com_hand, pBuffer:= ADR(qicsgp_buffer), szBuffer:= SIZEOF(qicsgp_buffer));			
	IF ComRead.xError THEN
		uiComState := 32767;
	END_IF
	IF ComRead.xDone THEN
		uiComState := 31;
		ComRead(xExecute := FALSE, hCom:= com_hand);
		position := find(qicsgp_buffer, 'OK');
		IF position > 0 THEN
			uiComState := 34;
		END_IF
	END_IF
	
	34: // write "AT+QIDEACT\r"     
	ComWrite(xExecute := TRUE,hCom:= com_hand,pBuffer:= ADR(qideact_cmd),szSize:=len(qideact_cmd));		
	IF ComWrite.xError THEN
		uiComState := 32767;
	END_IF
	IF ComWrite.xDone THEN
		ComWrite(xExecute := FALSE, hCom:= com_hand);
		uiComState := 35;
	END_IF
	
	35:
	ton_fb(IN := TRUE, PT := TIME#300MS);
	IF (ton_fb.Q) THEN
		ton_fb(IN := FALSE, PT := TIME#300MS);
		uiComState := 36;
	END_IF
	
	36:
	ComRead(xExecute := TRUE,hCom:= com_hand, pBuffer:= ADR(qicsgp_buffer), szBuffer:= SIZEOF(qicsgp_buffer));			
	IF ComRead.xError THEN
		uiComState := 32767;
	END_IF
	IF ComRead.xDone THEN
		uiComState := 34;
		ComRead(xExecute := FALSE, hCom:= com_hand);
		position := find(qicsgp_buffer, 'DEACT OK');
		IF position > 0 THEN
			uiComState := 37;
		END_IF
	END_IF
	
	37: // write "AT+QIREGAPP\r"     
	ComWrite(xExecute := TRUE,hCom:= com_hand,pBuffer:= ADR(qiregapp_cmd),szSize:=len(qiregapp_cmd));		
	IF ComWrite.xError THEN
		uiComState := 32767;
	END_IF
	IF ComWrite.xDone THEN
		ComWrite(xExecute := FALSE, hCom:= com_hand);
		uiComState := 38;
	END_IF
	
	38:
	ton_fb(IN := TRUE, PT := TIME#300MS);
	IF (ton_fb.Q) THEN
		ton_fb(IN := FALSE, PT := TIME#300MS);
		uiComState := 39;
	END_IF
	
	39:
	ComRead(xExecute := TRUE,hCom:= com_hand, pBuffer:= ADR(qiregapp_buffer), szBuffer:= SIZEOF(qiregapp_buffer));			
	IF ComRead.xError THEN
		uiComState := 32767;
	END_IF
	IF ComRead.xDone THEN
		uiComState := 37;
		ComRead(xExecute := FALSE, hCom:= com_hand);
		position := find(qiregapp_buffer, 'OK');
		IF position > 0 THEN
			uiComState := 40;
		END_IF
	END_IF
	
	40: // write "AT+QIACT\r"     
	ComWrite(xExecute := TRUE,hCom:= com_hand,pBuffer:= ADR(qiact_cmd),szSize:=len(qiact_cmd));		
	IF ComWrite.xError THEN
		uiComState := 32767;
	END_IF
	IF ComWrite.xDone THEN
		ComWrite(xExecute := FALSE, hCom:= com_hand);
		uiComState := 41;
	END_IF
	
	41:
	ton_fb(IN := TRUE, PT := TIME#300MS);
	IF (ton_fb.Q) THEN
		ton_fb(IN := FALSE, PT := TIME#300MS);
		uiComState := 42;
	END_IF
	
	42:
	ComRead(xExecute := TRUE,hCom:= com_hand, pBuffer:= ADR(qiact_buffer), szBuffer:= SIZEOF(qiact_buffer));			
	IF ComRead.xError THEN
		uiComState := 32767;
	END_IF
	IF ComRead.xDone THEN
		uiComState := 40;
		ComRead(xExecute := FALSE, hCom:= com_hand);
		position := find(qiact_buffer, 'OK');
		IF position > 0 THEN
			uiComState := 43;
		END_IF
	END_IF
	
	43: // write "AT+QILOCIP\r"     
	ComWrite(xExecute := TRUE,hCom:= com_hand,pBuffer:= ADR(qilocip_cmd),szSize:=len(qilocip_cmd));		
	IF ComWrite.xError THEN
		uiComState := 32767;
	END_IF
	IF ComWrite.xDone THEN
		ComWrite(xExecute := FALSE, hCom:= com_hand);
		uiComState := 44;
	END_IF
	
	44:
	ton_fb(IN := TRUE, PT := TIME#300MS);
	IF (ton_fb.Q) THEN
		ton_fb(IN := FALSE, PT := TIME#300MS);
		uiComState := 45;
	END_IF
	
	45:
	ComRead(xExecute := TRUE,hCom:= com_hand, pBuffer:= ADR(qilocip_buffer), szBuffer:= SIZEOF(qilocip_buffer));			
	IF ComRead.xError THEN
		uiComState := 32767;
	END_IF
	IF ComRead.xDone THEN
		uiComState := 46;
		ComRead(xExecute := FALSE, hCom:= com_hand);
		position := find(qilocip_buffer, 'ERROR');
		IF position > 0 THEN
			uiComState := 43;
		END_IF
	END_IF
	
	46:  // "AT+QNTP=\"s1a.time.edu.cn\"\r"
	ComWrite(xExecute := TRUE,hCom:= com_hand,pBuffer:= ADR(qntp_cmd),szSize:=len(qntp_cmd));		
	IF ComWrite.xError THEN
		uiComState := 32767;
	END_IF
	IF ComWrite.xDone THEN
		ComWrite(xExecute := FALSE, hCom:= com_hand);
		uiComState := 47;
	END_IF
	
	47:
	ton_fb(IN := TRUE, PT := TIME#300MS);
	IF (ton_fb.Q) THEN
		ton_fb(IN := FALSE, PT := TIME#300MS);
		uiComState := 48;
	END_IF
	
	48:
	ComRead(xExecute := TRUE,hCom:= com_hand, pBuffer:= ADR(qntp_buffer), szBuffer:= SIZEOF(qntp_buffer));			
	IF ComRead.xError THEN
		uiComState := 32767;
	END_IF
	IF ComRead.xDone THEN
		ComRead(xExecute := FALSE, hCom:= com_hand);
		uiComState := 49;
	END_IF

	49:  // "AT+QNITZ=1\r"
	ComWrite(xExecute := TRUE,hCom:= com_hand,pBuffer:= ADR(qnitz_cmd),szSize:=len(qnitz_cmd));		
	IF ComWrite.xError THEN
		uiComState := 32767;
	END_IF
	IF ComWrite.xDone THEN
		ComWrite(xExecute := FALSE, hCom:= com_hand);
		uiComState := 50;
	END_IF
	
	50:
	ton_fb(IN := TRUE, PT := TIME#300MS);
	IF (ton_fb.Q) THEN
		ton_fb(IN := FALSE, PT := TIME#300MS);
		uiComState := 51;
	END_IF
	
	51:
	ComRead(xExecute := TRUE,hCom:= com_hand, pBuffer:= ADR(qnitz_buffer), szBuffer:= SIZEOF(qnitz_buffer));			
	IF ComRead.xError THEN
		uiComState := 32767;
	END_IF
	IF ComRead.xDone THEN
		ComRead(xExecute := FALSE, hCom:= com_hand);
		uiComState := 52;
	END_IF
	
	52:  // "AT+CTZU=1\r"
	ComWrite(xExecute := TRUE,hCom:= com_hand,pBuffer:= ADR(ctzu_cmd),szSize:=len(ctzu_cmd));		
	IF ComWrite.xError THEN
		uiComState := 32767;
	END_IF
	IF ComWrite.xDone THEN
		ComWrite(xExecute := FALSE, hCom:= com_hand);
		uiComState := 53;
	END_IF
	
	53:
	ton_fb(IN := TRUE, PT := TIME#300MS);
	IF (ton_fb.Q) THEN
		ton_fb(IN := FALSE, PT := TIME#300MS);
		uiComState := 54;
	END_IF
	
	54:
	ComRead(xExecute := TRUE,hCom:= com_hand, pBuffer:= ADR(ctzu_buffer), szBuffer:= SIZEOF(ctzu_buffer));			
	IF ComRead.xError THEN
		uiComState := 32767;
	END_IF
	IF ComRead.xDone THEN
		ComRead(xExecute := FALSE, hCom:= com_hand);
		uiComState := 55;
	END_IF
	
	55:  // "AT+QLTS\r"
	ComWrite(xExecute := TRUE,hCom:= com_hand,pBuffer:= ADR(qlts_cmd),szSize:=len(qlts_cmd));		
	IF ComWrite.xError THEN
		uiComState := 32767;
	END_IF
	IF ComWrite.xDone THEN
		ComWrite(xExecute := FALSE, hCom:= com_hand);
		uiComState := 56;
	END_IF
	
	56:
	ton_fb(IN := TRUE, PT := TIME#300MS);
	IF (ton_fb.Q) THEN
		ton_fb(IN := FALSE, PT := TIME#300MS);
		uiComState := 57;
	END_IF
	
	57:
	ComRead(xExecute := TRUE,hCom:= com_hand, pBuffer:= ADR(qlts_buffer), szBuffer:= SIZEOF(qlts_buffer));			
	IF ComRead.xError THEN
		uiComState := 32767;
	END_IF
	IF ComRead.xDone THEN
		ComRead(xExecute := FALSE, hCom:= com_hand);
		uiComState := 58;
	END_IF
	
	58:  // "AT+CCLK?\r"
	ComWrite(xExecute := TRUE,hCom:= com_hand,pBuffer:= ADR(cclk_cmd),szSize:=len(cclk_cmd));		
	IF ComWrite.xError THEN
		uiComState := 32767;
	END_IF
	IF ComWrite.xDone THEN
		ComWrite(xExecute := FALSE, hCom:= com_hand);
		uiComState := 59;
	END_IF
	
	59:
	ton_fb(IN := TRUE, PT := TIME#300MS);
	IF (ton_fb.Q) THEN
		ton_fb(IN := FALSE, PT := TIME#300MS);
		uiComState := 60;
	END_IF
	
	60:
	ComRead(xExecute := TRUE,hCom:= com_hand, pBuffer:= ADR(cclk_buffer), szBuffer:= SIZEOF(cclk_buffer));			
	IF ComRead.xError THEN
		uiComState := 32767;
	END_IF
	IF ComRead.xDone THEN
		ComRead(xExecute := FALSE, hCom:= com_hand);
		NewDTS:=MID(qlts_buffer,20,11);    // NewDTS:=MID(cclk_buffer,20,11);
		NewDTSZH:=CONCAT('DT#20',left(NewDTS,2));
		year := ANY_TO_INT(left(NewDTS,2));
		NewDTSZH:=CONCAT(NewDTSZH,'-');	  
		NewDTSZH:=CONCAT(NewDTSZH,mid(NewDTS,2,4));	 
		NewDTSZH:=CONCAT(NewDTSZH,'-');	
		NewDTSZH:=CONCAT(NewDTSZH,mid(NewDTS,2,7));	
		NewDTSZH:=CONCAT(NewDTSZH,'-');	
		NewDTSZH:=CONCAT(NewDTSZH,mid(NewDTS,8,10));		  
		NewDT:=ANY_TO_DT(NewDTSZH);
		zone.iBias := -480;
		dtu_set_dt_fb(xExecute := FALSE);
		dtu_set_zone_fb(xExecute := FALSE);
		IF year >= 19 THEN
			uiComState := 62;
		ELSE
			uiComState := 63;	
		END_IF
	END_IF
	
	61:
	dtu_set_zone_fb(xExecute := TRUE, tziInfo := zone);			
	IF dtu_set_zone_fb.xError THEN
		uiComState := 32767;
	END_IF
	IF dtu_set_zone_fb.xDone THEN
		dtu_set_zone_fb(xExecute := FALSE);
		uiComState := 62;
	END_IF
	
	62:
	dtu_set_dt_fb(xExecute := TRUE, dtDateAndTime := STRING_TO_DT(NewDTSZH));		
	IF dtu_set_dt_fb.xError THEN
		uiComState := 32767;
	END_IF
	IF dtu_set_dt_fb.xDone THEN
		dtu_set_dt_fb(xExecute := FALSE);
		uiComState := 63;
		connect_cnt := 0;
	END_IF
	
	
	63: // write "AT+QIOPEN=\"UDP\",\"47.107.240.29\",123456\r"  
	qiopen_cmd := concat(qiopen_cmd, ip_addr);
	qiopen_cmd := concat(qiopen_cmd, '$",');
	qiopen_cmd := concat(qiopen_cmd, ANY_TO_STRING(port));
	qiopen_cmd := concat(qiopen_cmd, '$r');   
	ComWrite(xExecute := TRUE,hCom:= com_hand,pBuffer:= ADR(qiopen_cmd),szSize:=len(qiopen_cmd));		
	IF ComWrite.xError THEN
		uiComState := 32767;
	END_IF
	IF ComWrite.xDone THEN
		ComWrite(xExecute := FALSE, hCom:= com_hand);
		uiComState := 64;
	END_IF
	
	64:
	ton_fb(IN := TRUE, PT := TIME#300MS);
	IF (ton_fb.Q) THEN
		ton_fb(IN := FALSE, PT := TIME#300MS);
		uiComState := 65;
	END_IF
	
	65:
	ComRead(xExecute := TRUE,hCom:= com_hand, pBuffer:= ADR(qiopen_buffer), szBuffer:= SIZEOF(qiopen_buffer));			
	IF ComRead.xError THEN
		uiComState := 32767;
	END_IF
	IF ComRead.xDone THEN
		uiComState := 63;
		ComRead(xExecute := FALSE, hCom:= com_hand);
		position := find(qiopen_buffer, 'CONNECT OK');
		IF position > 0 THEN
			uiComState := 255;
		ELSE
			position := find(qiopen_buffer, 'ALREAY CONNECT');
			IF position > 0 THEN
				uiComState := 255;
			ELSE
				connect_cnt := connect_cnt + 1;
				IF connect_cnt > 50 THEN
					uiComState := 250;
					connect_cnt := 0;
				END_IF
			END_IF
		END_IF
	END_IF
	
	250:
	reset_gprs_fb.xExecute := TRUE;
	IF reset_gprs_fb.xDone THEN
		uiComState := 1;
	END_IF
	
	255:
		xDone := TRUE;
		
	32767:	
		xError := TRUE;
END_CASE

reset_gprs_fb();

END_FUNCTION_BLOCK

// MIC7001/Application/gprs_lib/reset_gprs
FUNCTION_BLOCK reset_gprs
VAR_INPUT
	xExecute:BOOL := FALSE;
END_VAR
VAR_OUTPUT
	xDone : BOOL := FALSE;
	xError :BOOL := FALSE;
	xBusy :BOOL := FALSE;
END_VAR
VAR
	iState :INT := 0;
	ton_fb :TON; 
END_VAR

IF NOT xExecute THEN
	iState := 0;
	xDone := FALSE;
	xBusy := FALSE;
	xError := FALSE;
	RETURN;
END_IF

CASE iState OF
0:
	xBusy := TRUE;
	set_gpio_value(129, 1);
	iState := 10;
	
10:
	ton_fb(IN := TRUE, PT := TIME#2000MS);
	IF (ton_fb.Q) THEN
		ton_fb(IN := FALSE, PT := TIME#2000MS);
		iState := 20;
	END_IF
	
20:
	set_gpio_value(129, 0);
	iState := 30;
	
30:
	ton_fb(IN := TRUE, PT := TIME#5000MS);
	IF (ton_fb.Q) THEN
		ton_fb(IN := FALSE, PT := TIME#5000MS);
		iState := 40;
	END_IF
	
40:
	iState := 255;	
	
255:
	xDone := TRUE;
	xBusy := FALSE;
32767:
	xError := TRUE;
END_CASE

END_FUNCTION_BLOCK

// MIC7001/Application/gprs_lib/Udp_Write
FUNCTION_BLOCK Udp_Write
VAR_INPUT
	xExecute :BOOL := FALSE;
	com :CAA.HANDLE;
	buffer: CAA.PVOID;
	size :CAA.SIZE;
END_VAR
VAR_OUTPUT
	xDone :BOOL := FALSE;
	xBusy :BOOL := FALSE;
	xError :BOOL := FALSE;
	atcState :INT;
END_VAR
VAR
	ComWrite: COM.Write;
	ComRead: COM.Read;	
	qisend_buffer :STRING := 'AT+QISEND='; 
	ton_fb :TON;  
	ack_buffer1 :STRING;
	ack_buffer2 :STRING;
	position :INT := -1;
	end_flag :ARRAY[0..1] OF BYTE;
	actionState :INT := 0;
	loop_count1 :INT := 0;
	loop_count2 :INT := 0;
	read_data_buffer: ARRAY[0..1499] OF BYTE;
END_VAR

IF NOT xExecute OR com = 0 THEN
	xDone := FALSE;
	xError := FALSE;
	xBusy := FALSE;
	actionState := 0;
	qisend_buffer := 'AT+QISEND='; 
	ComWrite(xExecute := FALSE);
	ComRead(xExecute := FALSE);
	RETURN;
END_IF

CASE actionState OF
0:
	ComRead(xExecute := TRUE,hCom:= com, pBuffer:= ADR(read_data_buffer), szBuffer:= SIZEOF(read_data_buffer));			
	IF ComRead.xError THEN
		ComRead(xExecute := FALSE);		
		actionState := 32767;
	END_IF
	IF ComRead.xDone THEN
		ComRead(xExecute := FALSE);			
		actionState := 1;
	END_IF

1:
	qisend_buffer := concat(qisend_buffer, ANY_TO_STRING(size));
	qisend_buffer := concat(qisend_buffer, '$r'); 
	actionState := 5;
	
5:
	ComWrite(xExecute := TRUE, hCom:= com, pBuffer:= ADR(qisend_buffer), szSize:= len(qisend_buffer));
	IF ComWrite.xError THEN
		actionState := 32767;
	END_IF
	IF ComWrite.xDone THEN
		actionState := 10;
		ComWrite(xExecute := FALSE, hCom:= com);	
	END_IF
	
10:
	ton_fb(IN := TRUE, PT := TIME#200MS);
	IF (ton_fb.Q) THEN
		ton_fb(IN := FALSE, PT := TIME#200MS);
		actionState := 20;
		ComRead(xExecute := FALSE);		
	END_IF
	
20:
	ComRead(xExecute := TRUE,hCom:= com, pBuffer:= ADR(ack_buffer1), szBuffer:= SIZEOF(ack_buffer1));			
	IF ComRead.xError THEN
		atcState := 32767;
	END_IF
	IF ComRead.xDone THEN
		
		position := find(ack_buffer1, '>');
		IF position > 0 THEN
			actionState := 30;
		ELSE
			actionState := 10;
		END_IF
		ComRead(xExecute := FALSE, hCom:= com);
		
		loop_count1 := loop_count1 + 1;
		IF loop_count1 > 50 THEN
			loop_count1 := 0;
			actionState := 32767;
		END_IF
	END_IF
	
30:
	ComWrite(xExecute := TRUE, hCom:= com, pBuffer:= buffer, szSize:= size);
	IF ComWrite.xError THEN
		actionState := 32767;
	END_IF
	IF ComWrite.xDone THEN
		actionState := 40;
		ComWrite(xExecute := FALSE, hCom:= com);	
	END_IF
	
40:
	end_flag[0] := 16#1A;
	ComWrite(xExecute := TRUE, hCom:= com, pBuffer:= ADR(end_flag), szSize:= 1);
	IF ComWrite.xError THEN
		actionState := 32767;
	END_IF
	IF ComWrite.xDone THEN
		actionState := 50;
		ComWrite(xExecute := FALSE, hCom:= com);	
	END_IF
	
50:
	ton_fb(IN := TRUE, PT := TIME#300MS);
	IF (ton_fb.Q) THEN
		ton_fb(IN := FALSE, PT := TIME#300MS);
		actionState := 60;
	END_IF
	
60:
	ComRead(xExecute := TRUE,hCom:= com, pBuffer:= ADR(ack_buffer2), szBuffer:= SIZEOF(ack_buffer2));			
	IF ComRead.xError THEN
		atcState := 32767;
	END_IF
	IF ComRead.xDone THEN
		position := find(ack_buffer2, 'SEND OK');
		IF position > 0 THEN
			actionState := 255;
		ELSE
			actionState := 50;
		END_IF
		ComRead(xExecute := FALSE, hCom:= com);
		loop_count2 := loop_count2 + 1;
		IF loop_count2 > 50 THEN
			loop_count2 := 0;
			actionState := 32767;
		END_IF
	END_IF
	
255:
	xDone := TRUE;
	xError := FALSE;
	xBusy := FALSE;
	actionState := 250;

	loop_count1 := 0;
	loop_count2 := 0; 
	ack_buffer1 := '';
	ack_buffer2 := '';
	qisend_buffer := 'AT+QISEND=';	
	
250:

32767:
	xDone := FALSE;
	xError := TRUE;
	xBusy := FALSE;
	actionState := 32700;

	loop_count1 := 0;
	loop_count2 := 0; 
	ack_buffer1 := '';
	ack_buffer2 := '';
	qisend_buffer := 'AT+QISEND=';	
	
32700:

END_CASE

END_FUNCTION_BLOCK

// MIC7001/Application/gprs_lib/UDP_Read
FUNCTION_BLOCK UDP_Read
VAR_INPUT
	xExecute:BOOL := FALSE;
	com :CAA.HANDLE;
	buffer: CAA.PVOID;
	rsize : CAA.SIZE;
END_VAR
VAR_OUTPUT
	xDone :BOOL := FALSE;
	xBusy :BOOL := FALSE;
	xError :BOOL := FALSE;
	size :CAA.SIZE;
	
END_VAR
VAR
	ton_fb :TON;  
	ComWrite: COM.Write;
	ComRead: COM.Read;	
	ack_buffer :STRING[1499];
	//ack_buffer :ARRAY[0..1499] OF BYTE;
	position :INT := -1;
	qird :STRING := 'AT+QIRD=0,1,0,1500$R';

	read_data_buffer: ARRAY[0..1499] OF BYTE;
	read_tmp_buffer: ARRAY[0..1499] OF BYTE;
	i :INT;
	read_num :INT;
	comma1 :INT;
	comma2 :INT;
	new_line :INT;
	data_len :INT := 0;
	//uchar *pos, *comma1, *comma2, *new_line;
	
	loop_count :INT := 0;
	loop_exit :INT := 0;
	
	del_atcState :INT;
	iStat :UINT := 0;
END_VAR

IF com = 0 OR NOT xExecute THEN
	xDone := FALSE;
	xError := FALSE;
	xBusy := FALSE;
	iStat := 0;
	position := -1;
	size := 0;
	ComRead(xExecute := FALSE);
	RETURN;
END_IF

CASE iStat OF
	0:
	ComRead(xExecute := TRUE,hCom:= com, pBuffer:= ADR(ack_buffer), szBuffer:= SIZEOF(ack_buffer));			
	IF ComRead.xError THEN
		ComRead(xExecute := FALSE, hCom:= com);
		iStat := 32767;
	END_IF
	
	IF ComRead.xDone THEN
		position := find(ack_buffer, '+QIRDI: 0,1,0');
		IF position > 0 THEN
			iStat := 2;
		ELSE
			iStat := 1;
		END_IF
		ComRead(xExecute := FALSE, hCom:= com);
		loop_count := loop_count + 1;
		IF loop_count > 20 THEN
			iStat := 2;
			loop_count := 0;
		END_IF
	END_IF
	
	1:
	ton_fb(IN := TRUE, PT := TIME#300MS);
	IF (ton_fb.Q) THEN
		ton_fb(IN := FALSE, PT := TIME#300MS);
		iStat := 0;
	END_IF
	
	2:
	ComWrite(xExecute := TRUE, hCom:= com, pBuffer:= ADR(qird), szSize:= len(qird));
	IF ComWrite.xError THEN
		iStat := 32767;
	END_IF
	
	IF ComWrite.xDone THEN
		iStat := 3;
		ComWrite(xExecute := FALSE, hCom:= com);	
	END_IF
	
	3:
	ton_fb(IN := TRUE, PT := TIME#300MS);
	IF (ton_fb.Q) THEN
		ton_fb(IN := FALSE, PT := TIME#300MS);
		iStat := 4;
	END_IF
	
	4:
	ComRead(xExecute := TRUE,hCom:= com, pBuffer:= ADR(read_data_buffer), szBuffer:= rsize);			
	IF ComRead.xError THEN
		iStat := 32767;
	END_IF
	IF ComRead.xDone THEN
		iStat := 5;
		read_num :=  ANY_TO_INT(ComRead.szSize);
		ComRead(xExecute := FALSE, hCom:= com);		
	END_IF
	
	5: //查找第一个逗号，第二次读取的时候，会返回OK，表示已经读完
	IF read_num = 6 THEN
		iStat := 0;
		loop_exit := loop_exit + 1;
		IF loop_exit > 1 THEN
			loop_exit := 0;
			iStat := 32767;
		END_IF
		RETURN;
	END_IF
	FOR i := 0 TO read_num - 1 BY 1 DO
		iStat := 32767;
		IF read_data_buffer[i] = 16#2C THEN
			comma1 := i;
			iStat := 6;
			RETURN;
		END_IF
	END_FOR;
	
	6: //查找第二个逗号
	FOR i := comma1 + 1 TO read_num - 1 BY 1 DO
		iStat := 32767;
		IF read_data_buffer[i] = 16#2C THEN
			comma2 := i;
			iStat := 7;
			RETURN;
		END_IF
	END_FOR;
	
	7: //查找回车换行
	FOR i := comma2 + 1 TO read_num - 1 BY 1 DO
		iStat := 32767;
		IF read_data_buffer[i] = 16#0D  AND read_data_buffer[i + 1] = 16#0A THEN
			new_line := i;
			iStat := 8;
			RETURN;
		END_IF
	END_FOR;
	
	8: // 获取数据长度
	FOR i := comma2 + 1 TO new_line - 1 BY 1 DO
		data_len := data_len *10 + read_data_buffer[i] - 16#30;
	END_FOR;

	iStat := 255;
	IF data_len > 0 THEN
		size := data_len;
		SysMemCpy(pDest:=buffer,pSrc:=ADR(read_data_buffer) + new_line + 2, udiCount:=data_len);
		
		data_len := 0;
		ack_buffer := '';
		loop_count := 0;
		read_num := 0;
		FOR i := 0 TO 1499 BY 1 DO
			read_data_buffer[i] := 0;
		END_FOR
	END_IF
	
	255:
		ComRead(xExecute := FALSE);
		xDone := TRUE;
		xBusy := FALSE;
		xError := FALSE;
		iStat := 256;
		
		data_len := 0;
		ack_buffer := '';
		loop_count := 0;
		read_num := 0;
		FOR i := 0 TO 1499 BY 1 DO
			read_data_buffer[i] := 0;
		END_FOR		
	256:
	
	32767:
		ComRead(xExecute := FALSE);
		xError := TRUE;
		xDone := FALSE;
		xBusy := FALSE;
		iStat := 32700;
		
		data_len := 0;
		ack_buffer := '';
		loop_count := 0;
		read_num := 0;
		FOR i := 0 TO 1499 BY 1 DO
			read_data_buffer[i] := 0;
		END_FOR		
	32700:
	
END_CASE

END_FUNCTION_BLOCK

// MIC7001/Application/GPRS/File_Read
FUNCTION_BLOCK File_Read
VAR_INPUT
	file_name :STRING;
END_VAR
VAR_OUTPUT
	sReadLine		: STRING;
	isRead          :BOOL := FALSE;	
END_VAR
VAR
	hfile			: CAA.HANDLE;
	FileOpen 		: File.Open;
	FileClose		: File.Close;
	FileRead		: File.Read;
	
	iState			: UINT := 0;	
	xError			: BOOL := FALSE;
END_VAR

 CASE iState OF
	0: // Open the file again, with read access.
	   isRead := false;
	   FileOpen(xExecute:= TRUE, sFileName:= file_name, xExclusive:= FALSE, eFileMode:= File.MODE.MREAD);
	   IF FileOpen.xDone = TRUE THEN
		   hfile := FileOpen.hFile;
		   FileOpen(xExecute:= FALSE);
		   iState := 1;
		   sReadLine := '';
	   ELSIF FileOpen.xError = TRUE THEN
		   iState:= 32767;
		   FileOpen(xExecute:= FALSE);
	   END_IF

	1: // Read the string from the file.
	   FileRead(xExecute:= TRUE, hFile:= hfile, pBuffer:= ADR(sReadLine), szBuffer:= SIZEOF(sReadLine));
	   IF FileRead.xDone = TRUE THEN
		   iState := 2;		   
		   sReadLine := MID(sReadLine, ANY_TO_INT(FileRead.szSize), 1);
		   FileRead(xExecute:= FALSE);
	   ELSIF FileRead.xError = TRUE THEN
		   iState:= 32767;
		   FileRead(xExecute:= FALSE);
	   END_IF 
	   
	 2: // Close that file.
	   FileClose(xExecute:= TRUE, hFile:= hfile);
	   IF FileClose.xDone = TRUE THEN
		   iState := 3;
		   FileClose(xExecute:= FALSE);
	   ELSIF FileClose.xError = TRUE THEN
		   iState:= 32767;
		   FileClose(xExecute:= FALSE);
	   END_IF
	   
	3: 	  
		isRead := TRUE;
		iState := 0;
		
	32767: 		
	
END_CASE

END_FUNCTION_BLOCK

// MIC7001/Application/gprs_lib/Com_Read
FUNCTION_BLOCK Com_Read
VAR_INPUT
	xExecute:BOOL := FALSE;
	com :CAA.HANDLE;
	wbuffer: CAA.PVOID;
	wsize :CAA.SIZE;	
	rbuffer: CAA.PVOID;
	rsize : CAA.SIZE;
END_VAR
VAR_OUTPUT
	xDone:BOOL := FALSE;
	xBusy:BOOL := FALSE;
	xError:BOOL := FALSE;
	size :CAA.SIZE;
END_VAR
VAR
	iState :INT;
	ton_fb :TON;  
	ComWrite: COM.Write;
	ComRead: COM.Read;	
	actionState :INT;
END_VAR

IF NOT xExecute THEN
	iState := 0;
	xDone := FALSE;
	xBusy := FALSE;
	xError := FALSE;
	size := 0;
	RETURN;
END_IF

CASE iState OF
0:
	size := 0;
	ComWrite(xExecute := TRUE, hCom:= com, pBuffer:= wbuffer, szSize:= wsize);
	IF ComWrite.xError THEN
		iState := 32767;
	END_IF
	IF ComWrite.xDone THEN
		iState := 10;
		ComWrite(xExecute := FALSE, hCom:= com);	
	END_IF
	xBusy := TRUE;
	
10:
	ton_fb(IN := TRUE, PT := TIME#300MS);
	IF (ton_fb.Q) THEN
		ton_fb(IN := FALSE, PT := TIME#300MS);
		iState := 20;
	END_IF
	
20:
	ComRead(xExecute := TRUE,hCom:= com, pBuffer:= rbuffer, szBuffer:= rsize);			
	IF ComRead.xError THEN
		iState := 32767;
	END_IF
	IF ComRead.xDone THEN
		iState := 255;
		size := ComRead.szSize;
		ComRead(xExecute := FALSE, hCom:= com);		
	END_IF
	
255:
	xDone := TRUE;
	xBusy := FALSE;
	
32767:
	xError := TRUE;
	
END_CASE

END_FUNCTION_BLOCK

// MIC7001/Application/GPRS/fb_get_iccid
FUNCTION_BLOCK fb_get_iccid
VAR_INPUT
	xExecute:BOOL := FALSE;
	m26_handle:CAA.HANDLE; 
END_VAR

VAR_OUTPUT
	iccid:STRING(32);
	xDone:BOOL := FALSE;
	xBusy :BOOL := FALSE;
	xError:BOOL := FALSE;
END_VAR

VAR
	iStat:UINT := 0;
	udp_handle :CAA.HANDLE; 
	accid_cmd :STRING := 'AT+ICCID$r';
	iccid_read_buffer :STRING(255);
	com_read :Com_Read;
	udp_init_fb: INT;
	size:CAA.SIZE;
	position :INT := -1;
	ICCID_HEAD:STRING := '+ICCID: ';
	timer01:ton;
END_VAR


IF NOT xExecute OR m26_handle = 0 THEN
	xDone := FALSE;
	xBusy := FALSE;
	xError := FALSE;
	iccid := '';
	iStat := 0;
	RETURN;
END_IF 		

IF iccid <> '' THEN  //已经读到了，不需再读
	xDone := TRUE;
	xBusy := FALSE;
	xError := FALSE;
	RETURN; 
END_IF

CASE iStat OF
0:
	com_read(xExecute := FALSE);
	iStat := 10;
	timer01(in := FALSE);
	com_read.xExecute := TRUE;
10:
	IF com_read.xDone THEN
		IF com_read.size > 0 THEN
			position := find(iccid_read_buffer, ICCID_HEAD);
			IF position > 0 THEN
				iccid := mid(iccid_read_buffer, 20, position + len(ICCID_HEAD));
				xDone := TRUE;
				iStat := 100;
			END_IF
		END_IF
	ELSIF com_read.xError THEN
		xDone := FALSE;
		iStat := 200;
	END_IF	
	timer01(in := NOT timer01.Q, pt := T#2S);
	IF timer01.Q THEN
		iStat := 0;
	END_IF
100:

200:

END_CASE

com_read(com:= m26_handle, wbuffer:= ADR(accid_cmd), wsize := len(accid_cmd), rbuffer := ADR(iccid_read_buffer), rsize := SIZEOF(iccid_read_buffer));

END_FUNCTION_BLOCK

// MIC7001/Application/GPRS/fb_get_lac
FUNCTION_BLOCK fb_get_lac
VAR_INPUT
	xExecute:BOOL := FALSE;
	m26_handle:CAA.HANDLE; 
END_VAR
VAR_OUTPUT
	lac:STRING(4) := '0000';
	ci :STRING(4) := '0000';
	xDone:BOOL := FALSE;
	xError:BOOL := FALSE;
END_VAR
VAR
	iStat:UINT := 0;
	udp_handle :CAA.HANDLE; 
	lac_set_cmd :STRING := 'AT+CREG=2$r';
	lac_get_cmd :STRING := 'AT+CREG?$r';
	lac_close_cmd :STRING := 'AT+CREG=0$r';
	lac_read_buffer :STRING(255);
	com_read :Com_Read;
	udp_init_fb: INT;
	size:CAA.SIZE;
	position :INT := -1;
	LACID_HEAD:STRING := '+CREG:';
	lac_str:STRING(8);
	ci_str:STRING(8);
	cntr: INT;
END_VAR


IF m26_handle = 0 THEN
	RETURN;
END_IF

IF NOT xExecute THEN
	xDone := FALSE;
	xError := FALSE;
	lac := '0000';
	ci := '0000';
	iStat := 0;
	
	RETURN;
END_IF 		

CASE iStat OF
0:
	com_read(xExecute := FALSE);
	com_read.wbuffer:= ADR(lac_set_cmd);
 	com_read.wsize := len(lac_set_cmd);
	com_read.xExecute := TRUE;	
	iStat := 5;
5:  //set m26 for lac and ci with command:  AT+CREG=2
	IF com_read.xDone THEN
		size := com_read.size;
		IF size > 0 THEN
			position := find(lac_read_buffer, 'OK');
			IF position > 0 THEN
				com_read(xExecute := FALSE);
				com_read.wbuffer:= ADR(lac_get_cmd);
				com_read.wsize := len(lac_get_cmd);
				com_read.xExecute := TRUE;				
				iStat := 10;
				cntr := 0;
			END_IF
		ELSE
			iStat := 0;
		END_IF
	ELSIF com_read.xError THEN
		xDone := FALSE;
	END_IF	

10:  //read lac and ci with command: AT+CREG?
	IF com_read.xDone THEN
		IF com_read.size > 0 THEN
			position := find(lac_read_buffer, LACID_HEAD);
			IF position > 0 THEN
				position := find(lac_read_buffer, '$"');
				IF position > 0 THEN
					lac := mid(lac_read_buffer, 4, position + 1);
					ci := mid(lac_read_buffer, 4, position + 8);
					iStat := 20;
					size := 0;
					com_read(xExecute := FALSE);
					com_read.wbuffer:= ADR(lac_close_cmd);
 					com_read.wsize := len(lac_close_cmd);
					com_read.xExecute := TRUE;
				END_IF
			ELSE
				iStat := 0;
			END_IF
		END_IF
		cntr := cntr + 1;
		IF cntr > 50 THEN
			iStat := 0;
		END_IF
	ELSIF com_read.xError THEN
		xDone := FALSE;
	END_IF	
	
20:  //close
	IF com_read.xDone THEN
		size := com_read.size;
		IF size > 0 THEN
			position := find(lac_read_buffer, 'OK');
			IF position > 0 THEN
				iStat := 100;
				xDone := TRUE;
			END_IF
		ELSE
			xDone := FALSE;
		END_IF
	ELSIF com_read.xError THEN
		xDone := FALSE;
	END_IF	
100: //ok

END_CASE

com_read(com:= m26_handle, rbuffer := ADR(lac_read_buffer), rsize := SIZEOF(lac_read_buffer));

END_FUNCTION_BLOCK
